// TIA Portal V19 export
ORGANIZATION_BLOCK "Rack or station failure"   // OB86, STL, RackOrStationFailure
TITLE = "Loss Of Rack Fault"
{ S7_Optimized_Access := 'FALSE' }
AUTHOR : RE
VERSION : 0.0
   VAR_TEMP
      OB86_EV_CLASS : Byte;   // 16#38/39 Event class 3
      OB86_FLT_ID : Byte;   // 16#C1/C4/C5, Fault identification code
      OB86_PRIORITY : Byte;   // 26/28 (Priority of 1 is lowest)
      OB86_OB_NUMBR : Byte;   // 86 (Organization block 86, OB86)
      OB86_RESERVED_1 : Byte;   // Reserved for system
      OB86_RESERVED_2 : Byte;   // Reserved for system
      OB86_MDL_ADDR : Word;   // Depending on fault identification code
      OB86_Z23 : DWord;   // see Context Help OB86
      OB86_DATE_TIME : Date_And_Time;   // Date and time OB86 started
      E_Param : DWord;
      RetVal : Int;
      DP_Slave_Nr : Int;
      Status : Array[0..1023] of Bool;
      Count : Int;
      Station_OK : Bool;
   END_VAR
BEGIN

NETWORK
TITLE = Wird bei DP-Stationsausfall und Rackfehler aktiviert
      AN    "DB_ANLAGE".IN.Watch_Profibus;  //keine Überwachung Profibus!
      BEC;

//DP-Slave Nummer
      L     #OB86_Z23.%W0;  //Nr. der DP Station (Bit 0-7 in OB86_Z23)
      AW    w#16#3ff;
      T     #DP_Slave_Nr;

//Fehler kommt/geht
      L     #OB86_EV_CLASS;
      L     16#39;  //kommendes Ereignis
      ==I;
      JC    kommt;

      L     #OB86_EV_CLASS;
      L     16#38;  //gehendes Ereignis
      ==I;
      JC    geht;

      BE;

NETWORK
TITLE = Fehler kommt
kommt:L     #OB86_FLT_ID;
      L     16#Cb;  //Ausfall einer DP-Station Code C4 Profinet CB
      <>I;
      BEC;

      L     #DP_Slave_Nr;
      SLD   3;
      LAR1;
      OPN   "DB_DP_Error";
      L     3;
      T     DBB [AR1, P#0.0];

      BE;

NETWORK
TITLE = Fehler geht
geht: L     #OB86_FLT_ID;
      L     16#Cb;  //Ausfall einer DP-Station gehendes Ereignis
      <>I;
      BEC;
      =     #Station_OK;

      L     #DP_Slave_Nr;
      SLD   3;
      LAR1;
      OPN   "DB_DP_Error";

      L     1;
      T     DBB [AR1, P#0.0];

// Check ob gestört
      CALL  DeviceStates
      ( LADDR   := "Local~PROFINET_IO-System",
        MODE    := 2,  // 2: IO-Devices/DP-Slaves gestört
        Ret_Val := #RetVal,
        STATE   := #Status
      );

//------------------------------------------------------------------------------
//Ergebnis abspeichern
      L     0;
      T     #Count;

      L     P##Status;
      LAR1;
      L     0;
retS: +AR1;

      AN    L [AR1, P#0.0];  //Laufendes Bit für Bus-Adresse
      JC    notS;

      L     #Count;
      T     "DB_DP_Error".HiAdr;  //höchste Adresse speichern
      SLD   3;
      LAR2;
      OPN   "DB_DP_Error";
      L     DBB [AR2, P#0.0];
      L     1;
      <>I;
      JC    notS;
      L     2;  //Station gestört
      T     DBB [AR2, P#0.0];

notS: L     #Count;
      +     1;
      T     #Count;
      L     1023;
      <D;
      L     P#0.1;
      JC    retS;
//------------------------------------------------------------------------------

      BE;
END_ORGANIZATION_BLOCK
